TYPE AliasOnlyThisProject :
STRUCT 
	systemTime : TIMESTRUCT;
	bValid : BOOL := true;
END_STRUCT
END_TYPE

(* stored: Version 1.1.0.1, ProductVersion 3.1.4024.12
   DUT AliasOnlyThisProject: Id {c1fa40a0-f430-476a-8fef-337194c5b0d5} *)
